TYPE CmpWorkStopMainLnSwSim :
STRUCT
	DBBypass: BOOL;
	ForceRFID: BOOL;
	TestRFIDData: DINT := 404;
	TestPuckData: DBGetOutputLane;
END_STRUCT
END_TYPE

(* stored: Version 1.1.0.1, ProductVersion 3.1.4024.6
   DUT CmpWorkStopMainLnSwSim: Id {eade88cd-7a92-4e00-b891-1b893d9a9e49} *)
